FUNCTION_BLOCK SELECTER (* Multi-purpose LED Flasher *)
  (* Standard: 61499 ITA *)
  (* Version 0.2, 2011-05-04, JHC, Holobloc Inc, Added XML line delimiters to Algorithms. *)
  (* Version 0.1, 2010-10-20, UnknownJHC, Holobloc Inc, Updated ECC transitions to 61499-1 Ed2 syntax. *)
  (* Version 0.0, 2004-01-09, JHC, Rockwell Automation, Copied from FLASHER4. *)
  (* Compiler header: package fb.rt.test; *)
  (* Compiler Java IBM VisualAge 3.0 *)
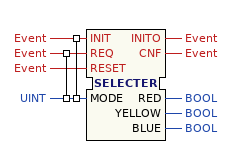
  EVENT_INPUT
    INIT WITH MODE; (* Initialization Request *)
    REQ WITH MODE; (* Update Request *)
    RESET;
  END_EVENT
  EVENT_OUTPUT
    INITO; (* Initialization Confirm *)
    CNF; (* Update Confirmation *)
  END_EVENT
  VAR_INPUT
    MODE : UINT; (* 0=FLASH_ALL,1=COUNT_UP,2=COUNT_DOWN,3=CHASE_UP,4=CHASE_DOWN *)
  END_VAR
  VAR_OUTPUT
    RED : BOOL;
    YELLOW : BOOL;
    BLUE : BOOL;
  END_VAR
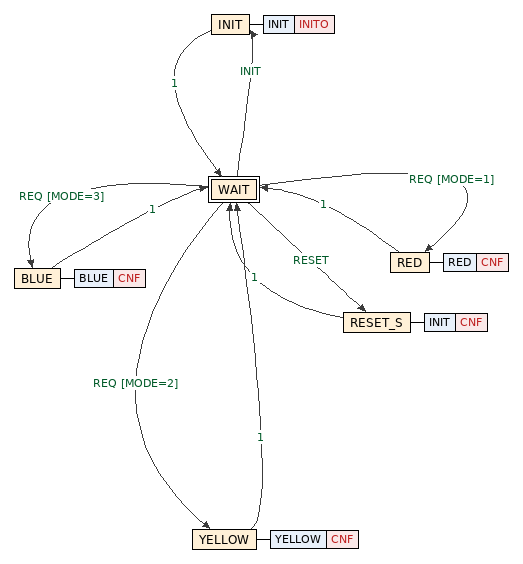
  EC_STATES
    WAIT;
    INIT : INIT -> INITO;
    RED : RED -> CNF;
    YELLOW : YELLOW -> CNF;
    BLUE : BLUE -> CNF;
    RESET_S : INIT -> CNF;
  END_STATES
  EC_TRANSITIONS
    WAIT TO INIT := INIT;
    WAIT TO RED := REQ [MODE=1];
    WAIT TO YELLOW := REQ [MODE=2];
    WAIT TO BLUE := REQ [MODE=3];
    INIT TO WAIT := 1;
    RED TO WAIT := 1;
    YELLOW TO WAIT := 1;
    BLUE TO WAIT := 1;
    WAIT TO RESET_S := RESET;
    RESET_S TO WAIT := 1;
  END_TRANSITIONS
  ALGORITHM INIT IN ST:
RED:=FALSE;
YELLOW:=FALSE;
BLUE:=FALSE;
  END_ALGORITHM
  ALGORITHM RED IN ST:
RED:=TRUE;
  END_ALGORITHM
  ALGORITHM YELLOW IN ST:
YELLOW:=TRUE;
  END_ALGORITHM
  ALGORITHM BLUE IN ST:
BLUE:=TRUE;
  END_ALGORITHM
END_FUNCTION_BLOCK
